FUNCTION_BLOCK InfoDataDC EXTENDS InfoDataBase
VAR
	_dcOutputShift AT %I* :   DINT;
	_dcInputShift AT %I* :   DINT;
END_VAR

PROPERTY DcInputShift : DINT
GET
DcInputShift := _dcInputShift;
END_GET
END_PROPERTY

PROPERTY DcOutputShift : DINT
GET
DcOutputShift := _dcOutputShift;
END_GET
END_PROPERTY

END_FUNCTION_BLOCK

(* stored: Version 1.1.0.1, ProductVersion 3.1.4024.9
   POU InfoDataDC: Id {bbbafae7-9efc-0662-3fad-233a957c2269}, SpecialFunc None
   Property DcInputShift: Id {f824b14c-5fc1-01e0-2c76-5b5da7bdd391}
   Get Get: Id {074db0cb-8cd2-0195-000b-3151dfac8fef}
   Property DcOutputShift: Id {9ff76fef-03e9-0170-1783-63874a9cac5e}
   Get Get: Id {a09fd5e3-d25b-042c-26e8-76ca37c9a088} *)
